PROGRAM POU_Output
VAR
END_VAR
//tower Lamp POU

// NETWORK 1

END_PROGRAM

(* stored: Version 1.1.0.1, ProductVersion 3.1.4024.0
   POU POU_Output: Id {8bcd174e-a6a1-4e07-8245-ad6cdc19d964}, SpecialFunc None *)
